TYPE E_HTTP_Request_Type :
(
	E_HTTP_Request_Type_GET := 0,
	E_HTTP_Request_Type_POST := 1
);
END_TYPE

(* stored: Version 1.1.0.1, ProductVersion 3.1.4020.12
   DUT E_HTTP_Request_Type: Id {5e0c8dce-6c90-4c8a-a445-f27ff32b6cf7} *)
